FUNCTION_BLOCK PUBLIC LINT_TO_TestSuite EXTENDS TcUnit.FB_TestSuite
VAR
END_VAR

Check_LINT_TO_BOOL_Max();
Check_LINT_TO_BOOL_Min();
Check_LINT_TO_BYTE_Max();
Check_LINT_TO_BYTE_Min();
Check_LINT_TO_BYTE_TooHigh();
Check_LINT_TO_BYTE_TooLow();
Check_LINT_TO_WORD_Max();
Check_LINT_TO_WORD_Min();
Check_LINT_TO_WORD_TooHigh();
Check_LINT_TO_WORD_TooLow();
Check_LINT_TO_DWORD_Max();
Check_LINT_TO_DWORD_Min();
Check_LINT_TO_DWORD_TooHigh();
Check_LINT_TO_DWORD_TooLow();
Check_LINT_TO_LWORD_Max();
Check_LINT_TO_LWORD_Min();
Check_LINT_TO_LWORD_TooLow();
Check_LINT_TO_SINT_Max();
Check_LINT_TO_SINT_Min();
Check_LINT_TO_SINT_TooHigh();
Check_LINT_TO_SINT_TooLow();
Check_LINT_TO_INT_Max();
Check_LINT_TO_INT_Min();
Check_LINT_TO_INT_TooHigh();
Check_LINT_TO_INT_TooLow();
Check_LINT_TO_DINT_Max();
Check_LINT_TO_DINT_Min();
Check_LINT_TO_DINT_TooHigh();
Check_LINT_TO_DINT_TooLow();
Check_LINT_TO_LINT_Max();
Check_LINT_TO_LINT_Min();
Check_LINT_TO_USINT_Max();
Check_LINT_TO_USINT_Min();
Check_LINT_TO_USINT_TooHigh();
Check_LINT_TO_USINT_TooLow();
Check_LINT_TO_UINT_Max();
Check_LINT_TO_UINT_Min();
Check_LINT_TO_UINT_TooHigh();
Check_LINT_TO_UINT_TooLow();
Check_LINT_TO_UDINT_Max();
Check_LINT_TO_UDINT_Min();
Check_LINT_TO_UDINT_TooHigh();
Check_LINT_TO_UDINT_TooLow();
Check_LINT_TO_ULINT_Max();
Check_LINT_TO_ULINT_Min();
Check_LINT_TO_ULINT_TooLow();
Check_LINT_TO_REAL_Max();
Check_LINT_TO_REAL_Min();
Check_LINT_TO_LREAL_Max();
Check_LINT_TO_LREAL_Min();
Check_LINT_TO_TIME_Max();
Check_LINT_TO_TIME_Min();
Check_LINT_TO_TIME_TooHigh();
Check_LINT_TO_TIME_TooLow();
Check_LINT_TO_TOD_Max();
Check_LINT_TO_TOD_Min();
Check_LINT_TO_TOD_TooHigh();
Check_LINT_TO_TOD_TooLow();
Check_LINT_TO_DATE_Max();
Check_LINT_TO_DATE_Min();
Check_LINT_TO_DATE_TooHigh();
Check_LINT_TO_DATE_TooLow();
Check_LINT_TO_DT_Max();
Check_LINT_TO_DT_Min();
Check_LINT_TO_DT_TooHigh();
Check_LINT_TO_DT_TooLow();
Check_LINT_TO_STRING_Max();
Check_LINT_TO_STRING_Min();

METHOD PUBLIC Check_LINT_TO_BOOL_Min
VAR
	value : LINT := DatatypeLimits.LINT_MIN_VALUE;
	actual : BOOL;
	converted : BOOL;
	equal : BOOL;
END_VAR
TEST('Check_LINT_TO_BOOL_Min');

// @TEST-RUN
converted := TryConvert_LINT_TO_Destination(value, actual);
equal := actual = LINT_TO_BOOL(value);

// @TEST-ASSERT
AssertTrue(Condition := equal, Message := 'Did not convert LINT to BOOL correctly');
AssertTrue(Condition := converted, Message := 'Did not report LINT to BOOL conversion was successful');

TEST_FINISHED();
END_METHOD

METHOD PUBLIC Check_LINT_TO_BOOL_Max
VAR
	value : LINT := DatatypeLimits.LINT_MAX_VALUE;
	actual : BOOL;
	converted : BOOL;
	equal : BOOL;
END_VAR
TEST('Check_LINT_TO_BOOL_Max');

// @TEST-RUN
converted := TryConvert_LINT_TO_Destination(value, actual);
equal := actual = LINT_TO_BOOL(value);

// @TEST-ASSERT
AssertTrue(Condition := equal, Message := 'Did not convert LINT to BOOL correctly');
AssertTrue(Condition := converted, Message := 'Did not report LINT to BOOL conversion was successful');

TEST_FINISHED();
END_METHOD

METHOD PUBLIC Check_LINT_TO_BYTE_Min
VAR
	value : LINT := DatatypeLimits.MIN_VALUE_OF_LINT_WHICH_CAN_BE_HELD_IN_A_BYTE;
	actual : BYTE;
	converted : BOOL;
	equal : BOOL;
END_VAR
TEST('Check_LINT_TO_BYTE_Min');

// @TEST-RUN
converted := TryConvert_LINT_TO_Destination(value, actual);
equal := actual = LINT_TO_BYTE(value);

// @TEST-ASSERT
AssertTrue(Condition := equal, Message := 'Did not convert LINT to BYTE correctly');
AssertTrue(Condition := converted, Message := 'Did not report LINT to BYTE conversion was successful');

TEST_FINISHED();
END_METHOD

METHOD PUBLIC Check_LINT_TO_BYTE_TooHigh
VAR
	value : LINT := DatatypeLimits.LINT_MAX_VALUE;
	actual : BYTE;
	converted : BOOL;
END_VAR
TEST('Check_LINT_TO_BYTE_TooHigh');

// @TEST-RUN
converted := TryConvert_LINT_TO_Destination(value, actual);

// @TEST-ASSERT
AssertFalse(Condition := converted, Message := 'Did not report LINT to BYTE conversion was prevented');

TEST_FINISHED();
END_METHOD

METHOD PUBLIC Check_LINT_TO_BYTE_TooLow
VAR
	value : LINT := DatatypeLimits.LINT_MIN_VALUE;
	actual : BYTE;
	converted : BOOL;
END_VAR
TEST('Check_LINT_TO_BYTE_TooLow');

// @TEST-RUN
converted := TryConvert_LINT_TO_Destination(value, actual);

// @TEST-ASSERT
AssertFalse(Condition := converted, Message := 'Did not report LINT to BYTE conversion was prevented');

TEST_FINISHED();
END_METHOD

METHOD PUBLIC Check_LINT_TO_BYTE_Max
VAR
	value : LINT := DatatypeLimits.MAX_VALUE_OF_LINT_WHICH_CAN_BE_HELD_IN_A_BYTE;
	actual : BYTE;
	converted : BOOL;
	equal : BOOL;
END_VAR
TEST('Check_LINT_TO_BYTE_Max');

// @TEST-RUN
converted := TryConvert_LINT_TO_Destination(value, actual);
equal := actual = LINT_TO_BYTE(value);

// @TEST-ASSERT
AssertTrue(Condition := equal, Message := 'Did not convert LINT to BYTE correctly');
AssertTrue(Condition := converted, Message := 'Did not report LINT to BYTE conversion was successful');

TEST_FINISHED();
END_METHOD

METHOD PUBLIC Check_LINT_TO_DATE_Min
VAR
	value : LINT := DatatypeLimits.MIN_VALUE_OF_LINT_WHICH_CAN_BE_HELD_IN_A_DATE;
	actual : DATE;
	converted : BOOL;
	equal : BOOL;
END_VAR
TEST('Check_LINT_TO_DATE_Min');

// @TEST-RUN
converted := TryConvert_LINT_TO_Destination(value, actual);
equal := actual = LINT_TO_DATE(value);

// @TEST-ASSERT
AssertTrue(Condition := equal, Message := 'Did not convert LINT to DATE correctly');
AssertTrue(Condition := converted, Message := 'Did not report LINT to DATE conversion was successful');

TEST_FINISHED();
END_METHOD

METHOD PUBLIC Check_LINT_TO_DATE_TooHigh
VAR
	value : LINT := DatatypeLimits.LINT_MAX_VALUE;
	actual : DATE;
	converted : BOOL;
END_VAR
TEST('Check_LINT_TO_DATE_TooHigh');

// @TEST-RUN
converted := TryConvert_LINT_TO_Destination(value, actual);

// @TEST-ASSERT
AssertFalse(Condition := converted, Message := 'Did not report LINT to DATE conversion was prevented');

TEST_FINISHED();
END_METHOD

METHOD PUBLIC Check_LINT_TO_DATE_TooLow
VAR
	value : LINT := DatatypeLimits.LINT_MIN_VALUE;
	actual : DATE;
	converted : BOOL;
END_VAR
TEST('Check_LINT_TO_DATE_TooLow');

// @TEST-RUN
converted := TryConvert_LINT_TO_Destination(value, actual);

// @TEST-ASSERT
AssertFalse(Condition := converted, Message := 'Did not report LINT to DATE conversion was prevented');

TEST_FINISHED();
END_METHOD

METHOD PUBLIC Check_LINT_TO_DATE_Max
VAR
	value : LINT := DatatypeLimits.MAX_VALUE_OF_LINT_WHICH_CAN_BE_HELD_IN_A_DATE;
	actual : DATE;
	converted : BOOL;
	equal : BOOL;
END_VAR
TEST('Check_LINT_TO_DATE_Max');

// @TEST-RUN
converted := TryConvert_LINT_TO_Destination(value, actual);
equal := actual = LINT_TO_DATE(value);

// @TEST-ASSERT
AssertTrue(Condition := equal, Message := 'Did not convert LINT to DATE correctly');
AssertTrue(Condition := converted, Message := 'Did not report LINT to DATE conversion was successful');

TEST_FINISHED();
END_METHOD

METHOD PUBLIC Check_LINT_TO_DINT_Min
VAR
	value : LINT := DatatypeLimits.MIN_VALUE_OF_LINT_WHICH_CAN_BE_HELD_IN_A_DINT;
	actual : DINT;
	converted : BOOL;
	equal : BOOL;
END_VAR
TEST('Check_LINT_TO_DINT_Min');

// @TEST-RUN
converted := TryConvert_LINT_TO_Destination(value, actual);
equal := actual = LINT_TO_DINT(value);

// @TEST-ASSERT
AssertTrue(Condition := equal, Message := 'Did not convert LINT to DINT correctly');
AssertTrue(Condition := converted, Message := 'Did not report LINT to DINT conversion was successful');

TEST_FINISHED();
END_METHOD

METHOD PUBLIC Check_LINT_TO_DINT_TooHigh
VAR
	value : LINT := DatatypeLimits.LINT_MAX_VALUE;
	actual : DINT;
	converted : BOOL;
END_VAR
TEST('Check_LINT_TO_DINT_TooHigh');

// @TEST-RUN
converted := TryConvert_LINT_TO_Destination(value, actual);

// @TEST-ASSERT
AssertFalse(Condition := converted, Message := 'Did not report LINT to DINT conversion was prevented');

TEST_FINISHED();
END_METHOD

METHOD PUBLIC Check_LINT_TO_DINT_TooLow
VAR
	value : LINT := DatatypeLimits.LINT_MIN_VALUE;
	actual : DINT;
	converted : BOOL;
END_VAR
TEST('Check_LINT_TO_DINT_TooLow');

// @TEST-RUN
converted := TryConvert_LINT_TO_Destination(value, actual);

// @TEST-ASSERT
AssertFalse(Condition := converted, Message := 'Did not report LINT to DINT conversion was prevented');

TEST_FINISHED();
END_METHOD

METHOD PUBLIC Check_LINT_TO_DINT_Max
VAR
	value : LINT := DatatypeLimits.MAX_VALUE_OF_LINT_WHICH_CAN_BE_HELD_IN_A_DINT;
	actual : DINT;
	converted : BOOL;
	equal : BOOL;
END_VAR
TEST('Check_LINT_TO_DINT_Max');

// @TEST-RUN
converted := TryConvert_LINT_TO_Destination(value, actual);
equal := actual = LINT_TO_DINT(value);

// @TEST-ASSERT
AssertTrue(Condition := equal, Message := 'Did not convert LINT to DINT correctly');
AssertTrue(Condition := converted, Message := 'Did not report LINT to DINT conversion was successful');

TEST_FINISHED();
END_METHOD

METHOD PUBLIC Check_LINT_TO_DT_Min
VAR
	value : LINT := DatatypeLimits.MIN_VALUE_OF_LINT_WHICH_CAN_BE_HELD_IN_A_DT;
	actual : DT;
	converted : BOOL;
	equal : BOOL;
END_VAR
TEST('Check_LINT_TO_DT_Min');

// @TEST-RUN
converted := TryConvert_LINT_TO_Destination(value, actual);
equal := actual = LINT_TO_DT(value);

// @TEST-ASSERT
AssertTrue(Condition := equal, Message := 'Did not convert LINT to DT correctly');
AssertTrue(Condition := converted, Message := 'Did not report LINT to DT conversion was successful');

TEST_FINISHED();
END_METHOD

METHOD PUBLIC Check_LINT_TO_DT_TooHigh
VAR
	value : LINT := DatatypeLimits.LINT_MAX_VALUE;
	actual : DT;
	converted : BOOL;
END_VAR
TEST('Check_LINT_TO_DT_TooHigh');

// @TEST-RUN
converted := TryConvert_LINT_TO_Destination(value, actual);

// @TEST-ASSERT
AssertFalse(Condition := converted, Message := 'Did not report LINT to DT conversion was prevented');

TEST_FINISHED();
END_METHOD

METHOD PUBLIC Check_LINT_TO_DT_TooLow
VAR
	value : LINT := DatatypeLimits.LINT_MIN_VALUE;
	actual : DT;
	converted : BOOL;
END_VAR
TEST('Check_LINT_TO_DT_TooLow');

// @TEST-RUN
converted := TryConvert_LINT_TO_Destination(value, actual);

// @TEST-ASSERT
AssertFalse(Condition := converted, Message := 'Did not report LINT to DT conversion was prevented');

TEST_FINISHED();
END_METHOD

METHOD PUBLIC Check_LINT_TO_DT_Max
VAR
	value : LINT := DatatypeLimits.MAX_VALUE_OF_LINT_WHICH_CAN_BE_HELD_IN_A_DT;
	actual : DT;
	converted : BOOL;
	equal : BOOL;
END_VAR
TEST('Check_LINT_TO_DT_Max');

// @TEST-RUN
converted := TryConvert_LINT_TO_Destination(value, actual);
equal := actual = LINT_TO_DT(value);

// @TEST-ASSERT
AssertTrue(Condition := equal, Message := 'Did not convert LINT to DT correctly');
AssertTrue(Condition := converted, Message := 'Did not report LINT to DT conversion was successful');

TEST_FINISHED();
END_METHOD

METHOD PUBLIC Check_LINT_TO_DWORD_Min
VAR
	value : LINT := DatatypeLimits.MIN_VALUE_OF_LINT_WHICH_CAN_BE_HELD_IN_A_DWORD;
	actual : DWORD;
	converted : BOOL;
	equal : BOOL;
END_VAR
TEST('Check_LINT_TO_DWORD_Min');

// @TEST-RUN
converted := TryConvert_LINT_TO_Destination(value, actual);
equal := actual = LINT_TO_DWORD(value);

// @TEST-ASSERT
AssertTrue(Condition := equal, Message := 'Did not convert LINT to DWORD correctly');
AssertTrue(Condition := converted, Message := 'Did not report LINT to DWORD conversion was successful');

TEST_FINISHED();
END_METHOD

METHOD PUBLIC Check_LINT_TO_DWORD_TooHigh
VAR
	value : LINT := DatatypeLimits.LINT_MAX_VALUE;
	actual : DWORD;
	converted : BOOL;
END_VAR
TEST('Check_LINT_TO_DWORD_TooHigh');

// @TEST-RUN
converted := TryConvert_LINT_TO_Destination(value, actual);

// @TEST-ASSERT
AssertFalse(Condition := converted, Message := 'Did not report LINT to DWORD conversion was prevented');

TEST_FINISHED();
END_METHOD

METHOD PUBLIC Check_LINT_TO_DWORD_TooLow
VAR
	value : LINT := DatatypeLimits.LINT_MIN_VALUE;
	actual : DWORD;
	converted : BOOL;
END_VAR
TEST('Check_LINT_TO_DWORD_TooLow');

// @TEST-RUN
converted := TryConvert_LINT_TO_Destination(value, actual);

// @TEST-ASSERT
AssertFalse(Condition := converted, Message := 'Did not report LINT to DWORD conversion was prevented');

TEST_FINISHED();
END_METHOD

METHOD PUBLIC Check_LINT_TO_DWORD_Max
VAR
	value : LINT := DatatypeLimits.MAX_VALUE_OF_LINT_WHICH_CAN_BE_HELD_IN_A_DWORD;
	actual : DWORD;
	converted : BOOL;
	equal : BOOL;
END_VAR
TEST('Check_LINT_TO_DWORD_Max');

// @TEST-RUN
converted := TryConvert_LINT_TO_Destination(value, actual);
equal := actual = LINT_TO_DWORD(value);

// @TEST-ASSERT
AssertTrue(Condition := equal, Message := 'Did not convert LINT to DWORD correctly');
AssertTrue(Condition := converted, Message := 'Did not report LINT to DWORD conversion was successful');

TEST_FINISHED();
END_METHOD

METHOD PUBLIC Check_LINT_TO_INT_Min
VAR
	value : LINT := DatatypeLimits.MIN_VALUE_OF_LINT_WHICH_CAN_BE_HELD_IN_A_INT;
	actual : INT;
	converted : BOOL;
	equal : BOOL;
END_VAR
TEST('Check_LINT_TO_INT_Min');

// @TEST-RUN
converted := TryConvert_LINT_TO_Destination(value, actual);
equal := actual = LINT_TO_INT(value);

// @TEST-ASSERT
AssertTrue(Condition := equal, Message := 'Did not convert LINT to INT correctly');
AssertTrue(Condition := converted, Message := 'Did not report LINT to INT conversion was successful');

TEST_FINISHED();
END_METHOD

METHOD PUBLIC Check_LINT_TO_INT_TooHigh
VAR
	value : LINT := DatatypeLimits.LINT_MAX_VALUE;
	actual : INT;
	converted : BOOL;
END_VAR
TEST('Check_LINT_TO_INT_TooHigh');

// @TEST-RUN
converted := TryConvert_LINT_TO_Destination(value, actual);

// @TEST-ASSERT
AssertFalse(Condition := converted, Message := 'Did not report LINT to INT conversion was prevented');

TEST_FINISHED();
END_METHOD

METHOD PUBLIC Check_LINT_TO_INT_TooLow
VAR
	value : LINT := DatatypeLimits.LINT_MIN_VALUE;
	actual : INT;
	converted : BOOL;
END_VAR
TEST('Check_LINT_TO_INT_TooLow');

// @TEST-RUN
converted := TryConvert_LINT_TO_Destination(value, actual);

// @TEST-ASSERT
AssertFalse(Condition := converted, Message := 'Did not report LINT to INT conversion was prevented');

TEST_FINISHED();
END_METHOD

METHOD PUBLIC Check_LINT_TO_INT_Max
VAR
	value : LINT := DatatypeLimits.MAX_VALUE_OF_LINT_WHICH_CAN_BE_HELD_IN_A_INT;
	actual : INT;
	converted : BOOL;
	equal : BOOL;
END_VAR
TEST('Check_LINT_TO_INT_Max');

// @TEST-RUN
converted := TryConvert_LINT_TO_Destination(value, actual);
equal := actual = LINT_TO_INT(value);

// @TEST-ASSERT
AssertTrue(Condition := equal, Message := 'Did not convert LINT to INT correctly');
AssertTrue(Condition := converted, Message := 'Did not report LINT to INT conversion was successful');

TEST_FINISHED();
END_METHOD

METHOD PUBLIC Check_LINT_TO_LINT_Min
VAR
	value : LINT := DatatypeLimits.LINT_MIN_VALUE;
	actual : LINT;
	converted : BOOL;
	equal : BOOL;
END_VAR
TEST('Check_LINT_TO_LINT_Min');

// @TEST-RUN
converted := TryConvert_LINT_TO_Destination(value, actual);
equal := actual = value;

// @TEST-ASSERT
AssertTrue(Condition := equal, Message := 'Did not convert LINT to LINT correctly');
AssertTrue(Condition := converted, Message := 'Did not report LINT to LINT conversion was successful');

TEST_FINISHED();
END_METHOD

METHOD PUBLIC Check_LINT_TO_LINT_Max
VAR
	value : LINT := DatatypeLimits.LINT_MAX_VALUE;
	actual : LINT;
	converted : BOOL;
	equal : BOOL;
END_VAR
TEST('Check_LINT_TO_LINT_Max');

// @TEST-RUN
converted := TryConvert_LINT_TO_Destination(value, actual);
equal := actual = value;

// @TEST-ASSERT
AssertTrue(Condition := equal, Message := 'Did not convert LINT to LINT correctly');
AssertTrue(Condition := converted, Message := 'Did not report LINT to LINT conversion was successful');

TEST_FINISHED();
END_METHOD

METHOD PUBLIC Check_LINT_TO_LREAL_Min
VAR
	value : LINT := DatatypeLimits.LINT_MIN_VALUE;
	actual : LREAL;
	converted : BOOL;
	equal : BOOL;
END_VAR
TEST('Check_LINT_TO_LREAL_Min');

// @TEST-RUN
converted := TryConvert_LINT_TO_Destination(value, actual);
equal := actual = LINT_TO_LREAL(value);

// @TEST-ASSERT
AssertTrue(Condition := equal, Message := 'Did not convert LINT to LREAL correctly');
AssertTrue(Condition := converted, Message := 'Did not report LINT to LREAL conversion was successful');

TEST_FINISHED();
END_METHOD

METHOD PUBLIC Check_LINT_TO_LREAL_Max
VAR
	value : LINT := DatatypeLimits.LINT_MAX_VALUE;
	actual : LREAL;
	converted : BOOL;
	equal : BOOL;
END_VAR
TEST('Check_LINT_TO_LREAL_Max');

// @TEST-RUN
converted := TryConvert_LINT_TO_Destination(value, actual);
equal := actual = LINT_TO_LREAL(value);

// @TEST-ASSERT
AssertTrue(Condition := equal, Message := 'Did not convert LINT to LREAL correctly');
AssertTrue(Condition := converted, Message := 'Did not report LINT to LREAL conversion was successful');

TEST_FINISHED();
END_METHOD

METHOD PUBLIC Check_LINT_TO_LWORD_Min
VAR
	value : LINT := DatatypeLimits.MIN_VALUE_OF_LINT_WHICH_CAN_BE_HELD_IN_A_LWORD;
	actual : LWORD;
	converted : BOOL;
	equal : BOOL;
END_VAR
TEST('Check_LINT_TO_LWORD_Min');

// @TEST-RUN
converted := TryConvert_LINT_TO_Destination(value, actual);
equal := actual = LINT_TO_LWORD(value);

// @TEST-ASSERT
AssertTrue(Condition := equal, Message := 'Did not convert LINT to LWORD correctly');
AssertTrue(Condition := converted, Message := 'Did not report LINT to LWORD conversion was successful');

TEST_FINISHED();
END_METHOD

METHOD PUBLIC Check_LINT_TO_LWORD_TooLow
VAR
	value : LINT := DatatypeLimits.LINT_MIN_VALUE;
	actual : LWORD;
	converted : BOOL;
END_VAR
TEST('Check_LINT_TO_LWORD_TooLow');

// @TEST-RUN
converted := TryConvert_LINT_TO_Destination(value, actual);

// @TEST-ASSERT
AssertFalse(Condition := converted, Message := 'Did not report LINT to LWORD conversion was prevented');

TEST_FINISHED();
END_METHOD

METHOD PUBLIC Check_LINT_TO_LWORD_Max
VAR
	value : LINT := DatatypeLimits.LINT_MAX_VALUE;
	actual : LWORD;
	converted : BOOL;
	equal : BOOL;
END_VAR
TEST('Check_LINT_TO_LWORD_Max');

// @TEST-RUN
converted := TryConvert_LINT_TO_Destination(value, actual);
equal := actual = LINT_TO_LWORD(value);

// @TEST-ASSERT
AssertTrue(Condition := equal, Message := 'Did not convert LINT to LWORD correctly');
AssertTrue(Condition := converted, Message := 'Did not report LINT to LWORD conversion was successful');

TEST_FINISHED();
END_METHOD

METHOD PUBLIC Check_LINT_TO_REAL_Min
VAR
	value : LINT := DatatypeLimits.LINT_MIN_VALUE;
	actual : REAL;
	converted : BOOL;
	equal : BOOL;
END_VAR
TEST('Check_LINT_TO_REAL_Min');

// @TEST-RUN
converted := TryConvert_LINT_TO_Destination(value, actual);
equal := actual = LINT_TO_REAL(value);

// @TEST-ASSERT
AssertTrue(Condition := equal, Message := 'Did not convert LINT to REAL correctly');
AssertTrue(Condition := converted, Message := 'Did not report LINT to REAL conversion was successful');

TEST_FINISHED();
END_METHOD

METHOD PUBLIC Check_LINT_TO_REAL_Max
VAR
	value : LINT := DatatypeLimits.LINT_MAX_VALUE;
	actual : REAL;
	converted : BOOL;
	equal : BOOL;
END_VAR
TEST('Check_LINT_TO_REAL_Max');

// @TEST-RUN
converted := TryConvert_LINT_TO_Destination(value, actual);
equal := actual = LINT_TO_REAL(value);

// @TEST-ASSERT
AssertTrue(Condition := equal, Message := 'Did not convert LINT to REAL correctly');
AssertTrue(Condition := converted, Message := 'Did not report LINT to REAL conversion was successful');

TEST_FINISHED();
END_METHOD

METHOD PUBLIC Check_LINT_TO_SINT_Min
VAR
	value : LINT := DatatypeLimits.MIN_VALUE_OF_LINT_WHICH_CAN_BE_HELD_IN_A_SINT;
	actual : SINT;
	converted : BOOL;
	equal : BOOL;
END_VAR
TEST('Check_LINT_TO_SINT_Min');

// @TEST-RUN
converted := TryConvert_LINT_TO_Destination(value, actual);
equal := actual = LINT_TO_SINT(value);

// @TEST-ASSERT
AssertTrue(Condition := equal, Message := 'Did not convert LINT to SINT correctly');
AssertTrue(Condition := converted, Message := 'Did not report LINT to SINT conversion was successful');

TEST_FINISHED();
END_METHOD

METHOD PUBLIC Check_LINT_TO_SINT_TooHigh
VAR
	value : LINT := DatatypeLimits.LINT_MAX_VALUE;
	actual : SINT;
	converted : BOOL;
END_VAR
TEST('Check_LINT_TO_SINT_TooHigh');

// @TEST-RUN
converted := TryConvert_LINT_TO_Destination(value, actual);

// @TEST-ASSERT
AssertFalse(Condition := converted, Message := 'Did not report LINT to SINT conversion was prevented');

TEST_FINISHED();
END_METHOD

METHOD PUBLIC Check_LINT_TO_SINT_TooLow
VAR
	value : LINT := DatatypeLimits.LINT_MIN_VALUE;
	actual : SINT;
	converted : BOOL;
END_VAR
TEST('Check_LINT_TO_SINT_TooLow');

// @TEST-RUN
converted := TryConvert_LINT_TO_Destination(value, actual);

// @TEST-ASSERT
AssertFalse(Condition := converted, Message := 'Did not report LINT to SINT conversion was prevented');

TEST_FINISHED();
END_METHOD

METHOD PUBLIC Check_LINT_TO_SINT_Max
VAR
	value : LINT := DatatypeLimits.MAX_VALUE_OF_LINT_WHICH_CAN_BE_HELD_IN_A_SINT;
	actual : SINT;
	converted : BOOL;
	equal : BOOL;
END_VAR
TEST('Check_LINT_TO_SINT_Max');

// @TEST-RUN
converted := TryConvert_LINT_TO_Destination(value, actual);
equal := actual = LINT_TO_SINT(value);

// @TEST-ASSERT
AssertTrue(Condition := equal, Message := 'Did not convert LINT to SINT correctly');
AssertTrue(Condition := converted, Message := 'Did not report LINT to SINT conversion was successful');

TEST_FINISHED();
END_METHOD

METHOD PUBLIC Check_LINT_TO_STRING_Min
VAR
	value : LINT := DatatypeLimits.LINT_MIN_VALUE;
	actual : STRING;
	converted : BOOL;
	equal : BOOL;
END_VAR
TEST('Check_LINT_TO_STRING_Min');

// @TEST-RUN
converted := TryConvert_LINT_TO_Destination(value, actual);
equal := actual = LINT_TO_STRING(value);

// @TEST-ASSERT
AssertTrue(Condition := equal, Message := 'Did not convert LINT to STRING correctly');
AssertTrue(Condition := converted, Message := 'Did not report LINT to STRING conversion was successful');

TEST_FINISHED();
END_METHOD

METHOD PUBLIC Check_LINT_TO_STRING_Max
VAR
	value : LINT := DatatypeLimits.LINT_MAX_VALUE;
	actual : STRING;
	converted : BOOL;
	equal : BOOL;
END_VAR
TEST('Check_LINT_TO_STRING_Max');

// @TEST-RUN
converted := TryConvert_LINT_TO_Destination(value, actual);
equal := actual = LINT_TO_STRING(value);

// @TEST-ASSERT
AssertTrue(Condition := equal, Message := 'Did not convert LINT to STRING correctly');
AssertTrue(Condition := converted, Message := 'Did not report LINT to STRING conversion was successful');

TEST_FINISHED();
END_METHOD

METHOD PUBLIC Check_LINT_TO_TIME_Min
VAR
	value : LINT := DatatypeLimits.MIN_VALUE_OF_LINT_WHICH_CAN_BE_HELD_IN_A_TIME;
	actual : TIME;
	converted : BOOL;
	equal : BOOL;
END_VAR
TEST('Check_LINT_TO_TIME_Min');

// @TEST-RUN
converted := TryConvert_LINT_TO_Destination(value, actual);
equal := actual = LINT_TO_TIME(value);

// @TEST-ASSERT
AssertTrue(Condition := equal, Message := 'Did not convert LINT to TIME correctly');
AssertTrue(Condition := converted, Message := 'Did not report LINT to TIME conversion was successful');

TEST_FINISHED();
END_METHOD

METHOD PUBLIC Check_LINT_TO_TIME_TooHigh
VAR
	value : LINT := DatatypeLimits.LINT_MAX_VALUE;
	actual : TIME;
	converted : BOOL;
END_VAR
TEST('Check_LINT_TO_TIME_TooHigh');

// @TEST-RUN
converted := TryConvert_LINT_TO_Destination(value, actual);

// @TEST-ASSERT
AssertFalse(Condition := converted, Message := 'Did not report LINT to TIME conversion was prevented');

TEST_FINISHED();
END_METHOD

METHOD PUBLIC Check_LINT_TO_TIME_TooLow
VAR
	value : LINT := DatatypeLimits.LINT_MIN_VALUE;
	actual : TIME;
	converted : BOOL;
END_VAR
TEST('Check_LINT_TO_TIME_TooLow');

// @TEST-RUN
converted := TryConvert_LINT_TO_Destination(value, actual);

// @TEST-ASSERT
AssertFalse(Condition := converted, Message := 'Did not report LINT to TIME conversion was prevented');

TEST_FINISHED();
END_METHOD

METHOD PUBLIC Check_LINT_TO_TIME_Max
VAR
	value : LINT := DatatypeLimits.MAX_VALUE_OF_LINT_WHICH_CAN_BE_HELD_IN_A_TIME;
	actual : TIME;
	converted : BOOL;
	equal : BOOL;
END_VAR
TEST('Check_LINT_TO_TIME_Max');

// @TEST-RUN
converted := TryConvert_LINT_TO_Destination(value, actual);
equal := actual = LINT_TO_TIME(value);

// @TEST-ASSERT
AssertTrue(Condition := equal, Message := 'Did not convert LINT to TIME correctly');
AssertTrue(Condition := converted, Message := 'Did not report LINT to TIME conversion was successful');

TEST_FINISHED();
END_METHOD

METHOD PUBLIC Check_LINT_TO_TOD_Min
VAR
	value : LINT := DatatypeLimits.MIN_VALUE_OF_LINT_WHICH_CAN_BE_HELD_IN_A_TOD;
	actual : TOD;
	converted : BOOL;
	equal : BOOL;
END_VAR
TEST('Check_LINT_TO_TOD_Min');

// @TEST-RUN
converted := TryConvert_LINT_TO_Destination(value, actual);
equal := actual = LINT_TO_TOD(value);

// @TEST-ASSERT
AssertTrue(Condition := equal, Message := 'Did not convert LINT to TOD correctly');
AssertTrue(Condition := converted, Message := 'Did not report LINT to TOD conversion was successful');

TEST_FINISHED();
END_METHOD

METHOD PUBLIC Check_LINT_TO_TOD_TooHigh
VAR
	value : LINT := DatatypeLimits.LINT_MAX_VALUE;
	actual : TOD;
	converted : BOOL;
END_VAR
TEST('Check_LINT_TO_TOD_TooHigh');

// @TEST-RUN
converted := TryConvert_LINT_TO_Destination(value, actual);

// @TEST-ASSERT
AssertFalse(Condition := converted, Message := 'Did not report LINT to TOD conversion was prevented');

TEST_FINISHED();
END_METHOD

METHOD PUBLIC Check_LINT_TO_TOD_TooLow
VAR
	value : LINT := DatatypeLimits.LINT_MIN_VALUE;
	actual : TOD;
	converted : BOOL;
END_VAR
TEST('Check_LINT_TO_TOD_TooLow');

// @TEST-RUN
converted := TryConvert_LINT_TO_Destination(value, actual);

// @TEST-ASSERT
AssertFalse(Condition := converted, Message := 'Did not report LINT to TOD conversion was prevented');

TEST_FINISHED();
END_METHOD

METHOD PUBLIC Check_LINT_TO_TOD_Max
VAR
	value : LINT := DatatypeLimits.MAX_VALUE_OF_LINT_WHICH_CAN_BE_HELD_IN_A_TOD;
	actual : TOD;
	converted : BOOL;
	equal : BOOL;
END_VAR
TEST('Check_LINT_TO_TOD_Max');

// @TEST-RUN
converted := TryConvert_LINT_TO_Destination(value, actual);
equal := actual = LINT_TO_TOD(value);

// @TEST-ASSERT
AssertTrue(Condition := equal, Message := 'Did not convert LINT to TOD correctly');
AssertTrue(Condition := converted, Message := 'Did not report LINT to TOD conversion was successful');

TEST_FINISHED();
END_METHOD

METHOD PUBLIC Check_LINT_TO_UDINT_Min
VAR
	value : LINT := DatatypeLimits.MIN_VALUE_OF_LINT_WHICH_CAN_BE_HELD_IN_A_UDINT;
	actual : UDINT;
	converted : BOOL;
	equal : BOOL;
END_VAR
TEST('Check_LINT_TO_UDINT_Min');

// @TEST-RUN
converted := TryConvert_LINT_TO_Destination(value, actual);
equal := actual = LINT_TO_UDINT(value);

// @TEST-ASSERT
AssertTrue(Condition := equal, Message := 'Did not convert LINT to UDINT correctly');
AssertTrue(Condition := converted, Message := 'Did not report LINT to UDINT conversion was successful');

TEST_FINISHED();
END_METHOD

METHOD PUBLIC Check_LINT_TO_UDINT_TooHigh
VAR
	value : LINT := DatatypeLimits.LINT_MAX_VALUE;
	actual : UDINT;
	converted : BOOL;
END_VAR
TEST('Check_LINT_TO_UDINT_TooHigh');

// @TEST-RUN
converted := TryConvert_LINT_TO_Destination(value, actual);

// @TEST-ASSERT
AssertFalse(Condition := converted, Message := 'Did not report LINT to UDINT conversion was prevented');

TEST_FINISHED();
END_METHOD

METHOD PUBLIC Check_LINT_TO_UDINT_TooLow
VAR
	value : LINT := DatatypeLimits.LINT_MIN_VALUE;
	actual : UDINT;
	converted : BOOL;
END_VAR
TEST('Check_LINT_TO_UDINT_TooLow');

// @TEST-RUN
converted := TryConvert_LINT_TO_Destination(value, actual);

// @TEST-ASSERT
AssertFalse(Condition := converted, Message := 'Did not report LINT to UDINT conversion was prevented');

TEST_FINISHED();
END_METHOD

METHOD PUBLIC Check_LINT_TO_UDINT_Max
VAR
	value : LINT := DatatypeLimits.MAX_VALUE_OF_LINT_WHICH_CAN_BE_HELD_IN_A_UDINT;
	actual : UDINT;
	converted : BOOL;
	equal : BOOL;
END_VAR
TEST('Check_LINT_TO_UDINT_Max');

// @TEST-RUN
converted := TryConvert_LINT_TO_Destination(value, actual);
equal := actual = LINT_TO_UDINT(value);

// @TEST-ASSERT
AssertTrue(Condition := equal, Message := 'Did not convert LINT to UDINT correctly');
AssertTrue(Condition := converted, Message := 'Did not report LINT to UDINT conversion was successful');

TEST_FINISHED();
END_METHOD

METHOD PUBLIC Check_LINT_TO_UINT_Min
VAR
	value : LINT := DatatypeLimits.MIN_VALUE_OF_LINT_WHICH_CAN_BE_HELD_IN_A_UINT;
	actual : UINT;
	converted : BOOL;
	equal : BOOL;
END_VAR
TEST('Check_LINT_TO_UINT_Min');

// @TEST-RUN
converted := TryConvert_LINT_TO_Destination(value, actual);
equal := actual = LINT_TO_UINT(value);

// @TEST-ASSERT
AssertTrue(Condition := equal, Message := 'Did not convert LINT to UINT correctly');
AssertTrue(Condition := converted, Message := 'Did not report LINT to UINT conversion was successful');

TEST_FINISHED();
END_METHOD

METHOD PUBLIC Check_LINT_TO_UINT_TooHigh
VAR
	value : LINT := DatatypeLimits.LINT_MAX_VALUE;
	actual : UINT;
	converted : BOOL;
END_VAR
TEST('Check_LINT_TO_UINT_TooHigh');

// @TEST-RUN
converted := TryConvert_LINT_TO_Destination(value, actual);

// @TEST-ASSERT
AssertFalse(Condition := converted, Message := 'Did not report LINT to UINT conversion was prevented');

TEST_FINISHED();
END_METHOD

METHOD PUBLIC Check_LINT_TO_UINT_TooLow
VAR
	value : LINT := DatatypeLimits.LINT_MIN_VALUE;
	actual : UINT;
	converted : BOOL;
END_VAR
TEST('Check_LINT_TO_UINT_TooLow');

// @TEST-RUN
converted := TryConvert_LINT_TO_Destination(value, actual);

// @TEST-ASSERT
AssertFalse(Condition := converted, Message := 'Did not report LINT to UINT conversion was prevented');

TEST_FINISHED();
END_METHOD

METHOD PUBLIC Check_LINT_TO_UINT_Max
VAR
	value : LINT := DatatypeLimits.MAX_VALUE_OF_LINT_WHICH_CAN_BE_HELD_IN_A_UINT;
	actual : UINT;
	converted : BOOL;
	equal : BOOL;
END_VAR
TEST('Check_LINT_TO_UINT_Max');

// @TEST-RUN
converted := TryConvert_LINT_TO_Destination(value, actual);
equal := actual = LINT_TO_UINT(value);

// @TEST-ASSERT
AssertTrue(Condition := equal, Message := 'Did not convert LINT to UINT correctly');
AssertTrue(Condition := converted, Message := 'Did not report LINT to UINT conversion was successful');

TEST_FINISHED();
END_METHOD

METHOD PUBLIC Check_LINT_TO_ULINT_Min
VAR
	value : LINT := DatatypeLimits.MIN_VALUE_OF_LINT_WHICH_CAN_BE_HELD_IN_A_ULINT;
	actual : ULINT;
	converted : BOOL;
	equal : BOOL;
END_VAR
TEST('Check_LINT_TO_ULINT_Min');

// @TEST-RUN
converted := TryConvert_LINT_TO_Destination(value, actual);
equal := actual = LINT_TO_ULINT(value);

// @TEST-ASSERT
AssertTrue(Condition := equal, Message := 'Did not convert LINT to ULINT correctly');
AssertTrue(Condition := converted, Message := 'Did not report LINT to ULINT conversion was successful');

TEST_FINISHED();
END_METHOD

METHOD PUBLIC Check_LINT_TO_ULINT_TooLow
VAR
	value : LINT := DatatypeLimits.LINT_MIN_VALUE;
	actual : ULINT;
	converted : BOOL;
END_VAR
TEST('Check_LINT_TO_ULINT_TooLow');

// @TEST-RUN
converted := TryConvert_LINT_TO_Destination(value, actual);

// @TEST-ASSERT
AssertFalse(Condition := converted, Message := 'Did not report LINT to ULINT conversion was prevented');

TEST_FINISHED();
END_METHOD

METHOD PUBLIC Check_LINT_TO_ULINT_Max
VAR
	value : LINT := DatatypeLimits.LINT_MAX_VALUE;
	actual : ULINT;
	converted : BOOL;
	equal : BOOL;
END_VAR
TEST('Check_LINT_TO_ULINT_Max');

// @TEST-RUN
converted := TryConvert_LINT_TO_Destination(value, actual);
equal := actual = LINT_TO_ULINT(value);

// @TEST-ASSERT
AssertTrue(Condition := equal, Message := 'Did not convert LINT to ULINT correctly');
AssertTrue(Condition := converted, Message := 'Did not report LINT to ULINT conversion was successful');

TEST_FINISHED();
END_METHOD

METHOD PUBLIC Check_LINT_TO_USINT_Min
VAR
	value : LINT := DatatypeLimits.MIN_VALUE_OF_LINT_WHICH_CAN_BE_HELD_IN_A_USINT;
	actual : USINT;
	converted : BOOL;
	equal : BOOL;
END_VAR
TEST('Check_LINT_TO_USINT_Min');

// @TEST-RUN
converted := TryConvert_LINT_TO_Destination(value, actual);
equal := actual = LINT_TO_USINT(value);

// @TEST-ASSERT
AssertTrue(Condition := equal, Message := 'Did not convert LINT to USINT correctly');
AssertTrue(Condition := converted, Message := 'Did not report LINT to USINT conversion was successful');

TEST_FINISHED();
END_METHOD

METHOD PUBLIC Check_LINT_TO_USINT_TooHigh
VAR
	value : LINT := DatatypeLimits.LINT_MAX_VALUE;
	actual : USINT;
	converted : BOOL;
END_VAR
TEST('Check_LINT_TO_USINT_TooHigh');

// @TEST-RUN
converted := TryConvert_LINT_TO_Destination(value, actual);

// @TEST-ASSERT
AssertFalse(Condition := converted, Message := 'Did not report LINT to USINT conversion was prevented');

TEST_FINISHED();
END_METHOD

METHOD PUBLIC Check_LINT_TO_USINT_TooLow
VAR
	value : LINT := DatatypeLimits.LINT_MIN_VALUE;
	actual : USINT;
	converted : BOOL;
END_VAR
TEST('Check_LINT_TO_USINT_TooLow');

// @TEST-RUN
converted := TryConvert_LINT_TO_Destination(value, actual);

// @TEST-ASSERT
AssertFalse(Condition := converted, Message := 'Did not report LINT to USINT conversion was prevented');

TEST_FINISHED();
END_METHOD

METHOD PUBLIC Check_LINT_TO_USINT_Max
VAR
	value : LINT := DatatypeLimits.MAX_VALUE_OF_LINT_WHICH_CAN_BE_HELD_IN_A_USINT;
	actual : USINT;
	converted : BOOL;
	equal : BOOL;
END_VAR
TEST('Check_LINT_TO_USINT_Max');

// @TEST-RUN
converted := TryConvert_LINT_TO_Destination(value, actual);
equal := actual = LINT_TO_USINT(value);

// @TEST-ASSERT
AssertTrue(Condition := equal, Message := 'Did not convert LINT to USINT correctly');
AssertTrue(Condition := converted, Message := 'Did not report LINT to USINT conversion was successful');

TEST_FINISHED();
END_METHOD

METHOD PUBLIC Check_LINT_TO_WORD_Min
VAR
	value : LINT := DatatypeLimits.MIN_VALUE_OF_LINT_WHICH_CAN_BE_HELD_IN_A_WORD;
	actual : WORD;
	converted : BOOL;
	equal : BOOL;
END_VAR
TEST('Check_LINT_TO_WORD_Min');

// @TEST-RUN
converted := TryConvert_LINT_TO_Destination(value, actual);
equal := actual = LINT_TO_WORD(value);

// @TEST-ASSERT
AssertTrue(Condition := equal, Message := 'Did not convert LINT to WORD correctly');
AssertTrue(Condition := converted, Message := 'Did not report LINT to WORD conversion was successful');

TEST_FINISHED();
END_METHOD

METHOD PUBLIC Check_LINT_TO_WORD_TooHigh
VAR
	value : LINT := DatatypeLimits.LINT_MAX_VALUE;
	actual : WORD;
	converted : BOOL;
END_VAR
TEST('Check_LINT_TO_WORD_TooHigh');

// @TEST-RUN
converted := TryConvert_LINT_TO_Destination(value, actual);

// @TEST-ASSERT
AssertFalse(Condition := converted, Message := 'Did not report LINT to WORD conversion was prevented');

TEST_FINISHED();
END_METHOD

METHOD PUBLIC Check_LINT_TO_WORD_TooLow
VAR
	value : LINT := DatatypeLimits.LINT_MIN_VALUE;
	actual : WORD;
	converted : BOOL;
END_VAR
TEST('Check_LINT_TO_WORD_TooLow');

// @TEST-RUN
converted := TryConvert_LINT_TO_Destination(value, actual);

// @TEST-ASSERT
AssertFalse(Condition := converted, Message := 'Did not report LINT to WORD conversion was prevented');

TEST_FINISHED();
END_METHOD

METHOD PUBLIC Check_LINT_TO_WORD_Max
VAR
	value : LINT := DatatypeLimits.MAX_VALUE_OF_LINT_WHICH_CAN_BE_HELD_IN_A_WORD;
	actual : WORD;
	converted : BOOL;
	equal : BOOL;
END_VAR
TEST('Check_LINT_TO_WORD_Max');

// @TEST-RUN
converted := TryConvert_LINT_TO_Destination(value, actual);
equal := actual = LINT_TO_WORD(value);

// @TEST-ASSERT
AssertTrue(Condition := equal, Message := 'Did not convert LINT to WORD correctly');
AssertTrue(Condition := converted, Message := 'Did not report LINT to WORD conversion was successful');

TEST_FINISHED();
END_METHOD

END_FUNCTION_BLOCK

(* stored: Version 1.1.0.1, ProductVersion 3.1.4024.12
   POU LINT_TO_TestSuite: Id {8810f156-54d7-408e-82b1-477d2c607c26}, SpecialFunc None
   Method Check_LINT_TO_BOOL_Min: Id {42c0fc53-df6f-4105-b75b-4ec7d61de7e0}
   Method Check_LINT_TO_BOOL_Max: Id {e26bf448-a808-43d5-944b-4b73a3845b05}
   Method Check_LINT_TO_BYTE_Min: Id {5ccf301e-c08f-4938-95fd-96db8b58c73c}
   Method Check_LINT_TO_BYTE_TooHigh: Id {70c7fc76-f628-463e-be3d-916ae53dfb10}
   Method Check_LINT_TO_BYTE_TooLow: Id {c022a252-fa42-4172-8a7f-87e03659d4e3}
   Method Check_LINT_TO_BYTE_Max: Id {61dc699b-2acb-4d58-9821-350f8bb1aeab}
   Method Check_LINT_TO_DATE_Min: Id {6e4b2a9f-a2eb-43dd-8a6f-31537b5d3582}
   Method Check_LINT_TO_DATE_TooHigh: Id {e63af9b5-fa15-4296-a3df-767d9697f8ab}
   Method Check_LINT_TO_DATE_TooLow: Id {539404e7-37ac-4f92-a9e9-07b508b37e52}
   Method Check_LINT_TO_DATE_Max: Id {544b2ef5-6c10-4d32-be91-7e6b7be83585}
   Method Check_LINT_TO_DINT_Min: Id {1d67ec21-5c0f-4170-8aa8-60b328e5f79b}
   Method Check_LINT_TO_DINT_TooHigh: Id {cfd2aeec-e06a-4f3e-a518-5417baca01e5}
   Method Check_LINT_TO_DINT_TooLow: Id {ea77ea2c-55db-4de0-8623-f2bebc9b633c}
   Method Check_LINT_TO_DINT_Max: Id {5d386188-5ffd-4aec-b216-fda18d8efca3}
   Method Check_LINT_TO_DT_Min: Id {648f62d0-2fbf-4e99-91be-e68dd7b10fcc}
   Method Check_LINT_TO_DT_TooHigh: Id {d017fcd4-0b63-46b6-a0b7-9871ec32b4ad}
   Method Check_LINT_TO_DT_TooLow: Id {e05d3e15-20ba-4b81-a94e-af0f1546e0a3}
   Method Check_LINT_TO_DT_Max: Id {c96c58d2-d95f-41ff-9d51-08abfbf8efab}
   Method Check_LINT_TO_DWORD_Min: Id {f2cab39c-c7e3-43bc-8d71-d183983ba3d8}
   Method Check_LINT_TO_DWORD_TooHigh: Id {a1a0be18-fd94-49e4-98d1-a75c9cfa80b2}
   Method Check_LINT_TO_DWORD_TooLow: Id {44e97f1e-eb77-40bb-aaaf-1b44c512f662}
   Method Check_LINT_TO_DWORD_Max: Id {7f345cf3-2892-484e-95e9-4fe631f2bb12}
   Method Check_LINT_TO_INT_Min: Id {50346f33-0eff-4e6f-a036-f554e7fc7962}
   Method Check_LINT_TO_INT_TooHigh: Id {976bde4f-6a23-46cc-89b9-3ed85d5451da}
   Method Check_LINT_TO_INT_TooLow: Id {ee8101bf-eae8-4e07-8f03-bea582e416df}
   Method Check_LINT_TO_INT_Max: Id {a96e57e8-3785-4a75-a6b7-825c12ec7fb2}
   Method Check_LINT_TO_LINT_Min: Id {97cd8e49-dc1d-4123-a5c7-8940926e5747}
   Method Check_LINT_TO_LINT_Max: Id {08f2d8e7-22c0-48fe-8b5d-fdb4b463b6ea}
   Method Check_LINT_TO_LREAL_Min: Id {3bbf1a0b-6d4a-436f-81fd-52b9fc79b997}
   Method Check_LINT_TO_LREAL_Max: Id {c43d2abe-025b-4f17-82c9-bad9c9866dec}
   Method Check_LINT_TO_LWORD_Min: Id {60fec2f4-09aa-4a23-8dad-ad5f0bfc7c94}
   Method Check_LINT_TO_LWORD_TooLow: Id {7d8da66b-52d6-4555-a6e9-c96199377ed1}
   Method Check_LINT_TO_LWORD_Max: Id {41085455-b6f0-43b9-8b07-af75b7839aad}
   Method Check_LINT_TO_REAL_Min: Id {5072b32e-36cf-40a2-8779-501ff6e33ab7}
   Method Check_LINT_TO_REAL_Max: Id {d272aa93-4192-4fe5-9eed-cedef6f8032d}
   Method Check_LINT_TO_SINT_Min: Id {96c6411a-6bd8-4bdf-a402-5221d05c3c8a}
   Method Check_LINT_TO_SINT_TooHigh: Id {d4b83c48-f93b-469a-81cb-0ac74b282104}
   Method Check_LINT_TO_SINT_TooLow: Id {12737fd9-1411-4321-bace-96a59609c76d}
   Method Check_LINT_TO_SINT_Max: Id {81cd1547-8390-428e-9c65-ad74c9068bc5}
   Method Check_LINT_TO_STRING_Min: Id {cfd6e4f0-8d47-48cb-8157-9348c8b1733c}
   Method Check_LINT_TO_STRING_Max: Id {01b4a72c-c1e0-4a84-b047-873d174fc9a6}
   Method Check_LINT_TO_TIME_Min: Id {2aa2f220-ab25-45c4-89d0-fa2aca878314}
   Method Check_LINT_TO_TIME_TooHigh: Id {41b0a828-9a7a-49d7-a4d5-0b441c2233e8}
   Method Check_LINT_TO_TIME_TooLow: Id {0a22d689-4d35-46a4-82d2-c87548cbfcc4}
   Method Check_LINT_TO_TIME_Max: Id {55650074-f23f-41b3-bd31-9b91346ff1f0}
   Method Check_LINT_TO_TOD_Min: Id {92c4ad07-5e37-48e5-9c43-e6c0a8a24669}
   Method Check_LINT_TO_TOD_TooHigh: Id {180abb5a-ae97-4126-8eb8-9eb238e278c7}
   Method Check_LINT_TO_TOD_TooLow: Id {ca4c9459-b42c-41be-bdf7-8b0c430c5c60}
   Method Check_LINT_TO_TOD_Max: Id {e422d51a-8f04-4d65-a35d-3435485bbd71}
   Method Check_LINT_TO_UDINT_Min: Id {f96de0ce-0e98-4719-b0c6-f72bd41a03b0}
   Method Check_LINT_TO_UDINT_TooHigh: Id {aee4ace3-6c5d-4c21-aa6a-b07c33f6483c}
   Method Check_LINT_TO_UDINT_TooLow: Id {e993218f-0f10-4ced-9e39-12e655d9b228}
   Method Check_LINT_TO_UDINT_Max: Id {d605a80b-ea2d-4db0-9eb6-cab82dc0b4d9}
   Method Check_LINT_TO_UINT_Min: Id {dde52459-9e59-4cb9-b3c5-bb7e08c66251}
   Method Check_LINT_TO_UINT_TooHigh: Id {b7216e73-ce48-4c22-8190-a057abf6c492}
   Method Check_LINT_TO_UINT_TooLow: Id {8ec175bb-d9d9-455e-91ae-32a0319d7352}
   Method Check_LINT_TO_UINT_Max: Id {ad7ac0bc-d499-4f9c-985f-7a1a91f137e0}
   Method Check_LINT_TO_ULINT_Min: Id {1db82dd7-d79e-4d8f-8fbb-9138aaf42fa4}
   Method Check_LINT_TO_ULINT_TooLow: Id {f2a98633-30de-43f3-9d39-fbda68e8eba9}
   Method Check_LINT_TO_ULINT_Max: Id {deb971c7-867c-4ca9-8bad-ac1aef190bf5}
   Method Check_LINT_TO_USINT_Min: Id {deee47e6-6138-4f62-8609-839283ca6df9}
   Method Check_LINT_TO_USINT_TooHigh: Id {9a7a9cfe-ab83-427e-925d-08670c917270}
   Method Check_LINT_TO_USINT_TooLow: Id {97ad46db-cb90-4d3b-8020-acea9e3a9e7a}
   Method Check_LINT_TO_USINT_Max: Id {8508483c-5d39-464d-a5d7-4f2bdf3f9e11}
   Method Check_LINT_TO_WORD_Min: Id {c68d42f6-322e-4c38-949a-a73c054f0525}
   Method Check_LINT_TO_WORD_TooHigh: Id {8c35b95e-2907-475e-8d84-1f8ce051c1b2}
   Method Check_LINT_TO_WORD_TooLow: Id {fa569f72-4c46-4def-86d7-8cc2c782ec2d}
   Method Check_LINT_TO_WORD_Max: Id {1cd4d22e-7f41-4af8-8c4f-e75e51fd541c} *)
